PROGRAM MAIN
VAR
	bEnable: BOOL;
	bStart : BOOL;
END_VAR

bEnable := bStart;

END_PROGRAM

(* stored: Version 1.1.0.1, ProductVersion 3.1.4024.12
   POU MAIN: Id {69050987-6d20-4df5-a8b6-664f154c8c17}, SpecialFunc None *)
